// TwinCAT 3 PLC project PID_Projekt
// ProgramVersion: 3.1.4023.0
// libraries:
//   Tc2_ControllerToolbox, * (Beckhoff Automation GmbH)
//   Tc2_MC2, * (Beckhoff Automation GmbH)
//   Tc2_Standard, * (Beckhoff Automation GmbH)
//   Tc2_System, * (Beckhoff Automation GmbH)
//   Tc3_Module, * (Beckhoff Automation GmbH)
// project tree:
//   DUTs/ state.TcDUT
//   / GlobalTextList.TcGTLO, PID_Task.TcTTO, PlcTask.TcTTO
//   GVLs/ GVL.TcGVL
//   POUs/ MAIN.TcPOU
//   POUs/PID/ PID_Call.TcPOU, PRG_FB_CTRL_D.TcPOU, PRG_FB_CTRL_I.TcPOU, PRG_FB_CTRL_P.TcPOU
// real-time tasks:
//   TASK PlcTask: cycle T#1ms, priority 2, ADS port 350
//   TASK PID_Task: cycle T#10ms, priority 3, ADS port 351
// motion (NC):
//   TASK NC-Task 1 SAF: cycle T#1ms, priority 1, ADS port 501
//   TASK NC-Task 1 SVB: cycle T#10ms, priority 8, ADS port 511
//   AXIS Achse 1 (id 1) // MyAxis
//     Dynamic: Acceleration=3000, Deceleration=500
//     OtherSettings: AllowMotionCmdToSlave=true
//     encoder EncType=1
//     drive DrvType=5
//       Analog: TorqueSetpointScale=10, ScaleFactorActTorque=0.1
//       TimeComp: TaskDelayCycles=1
//     controller CtrType=1
//       CtrPara: PriorControlFactor=1
//         Observer: BandWidth=20
// variable links:
//   PID_Projekt/PID_Projekt Instance <-> NC-Task 1 SAF/Axes/Achse 1
//     PlcTask Inputs/MAIN.axis.NcToPlc <-> Outputs/ToPlc
//     PlcTask Outputs/MAIN.axis.PlcToNc <-> Inputs/FromPlc

CONFIGURATION PID_Projekt
    RESOURCE PLC ON TwinCAT3
        TASK PID_Task(INTERVAL := T#10ms, PRIORITY := 3);
        TASK PlcTask(INTERVAL := T#1ms, PRIORITY := 2);
        PROGRAM PID_Call WITH PID_Task : PID_Call;
        PROGRAM MAIN WITH PlcTask : MAIN;
    END_RESOURCE
END_CONFIGURATION

// ---- DUTs/state.TcDUT
TYPE state :
(
	INIT,
	POWER_ON,
	MOVE_ON,
	//MOVE_ON_NEWTARGETPOSITION,
	ERROR,
	P_RESET
)UDINT;
END_TYPE

// ---- GVLs/GVL.TcGVL
{attribute 'qualified_only'}
VAR_GLOBAL
	Signal: LREAL;
	Position: LREAL;
	Velocity: LREAL;
	Sollkraft: LREAL := 1;
	ErrorTerm: LREAL;
	PID_Output: LREAL;
	P_Regler: LREAL;
	I_Regler: LREAL;
	D_Regler: LREAL;
END_VAR

// ---- POUs/PID/PID_Call.TcPOU
PROGRAM PID_Call
VAR
	Simulation: BOOL := 0;
	Stoerungen: LREAL;
	SteadyState: BOOL := 0;
	D_Regler_Switch: BOOL := 1;
	I_Regler_Switch: BOOL := 1;
	Kp: LREAL;
	Satuaration_Check_LimMax: LREAL := 0.5;
	Satuaration_Check_LimMin: LREAL := -0.5;
	Not_Equal_Block: BOOL;
	Equal_Block: BOOL;
	PID_Output_after_S_check: LREAL;
	Drand: DRAND;
	PID_OUT_LimMin: LREAL := -0.9;
	PID_OUT_LimMax: LREAL := 0.9;
END_VAR

//*********Sensor
Drand(Seed:=0);
Stoerungen := (Drand.Num-0.5)*0.02;
GVL.Position := GVL.Position * (1+Stoerungen);
//GVL.Signal := GVL.Position;

//*********Error Term from Feedback Path
Drand(Seed:=0);	
Stoerungen := (Drand.Num-0.5)*0.02;
GVL.Signal := GVL.Position * (1+Stoerungen);
GVL.ErrorTerm := GVL.Sollkraft - GVL.Signal;

IF GVL.Position<(GVL.Sollkraft+0.015) AND GVL.Position>(GVL.Sollkraft-0.015) THEN
	SteadyState :=1;
ELSE SteadyState :=0;
END_IF

IF Simulation = 1 THEN
	GVL.ErrorTerm := GVL.Sollkraft - GVL.Signal * (1+(Drand.Num-0.5)*1);
END_IF

IF SteadyState = 0 THEN
	GVL.ErrorTerm := GVL.Sollkraft - GVL.Position;
	D_Regler_Switch := 0;
ELSE
//	GVL.ErrorTerm := GVL.Sollkraft - GVL.Signal;
	D_Regler_Switch := 1;
END_IF

//************I-Regler
PRG_FB_CTRL_P();

//************I-Regler
IF I_Regler_Switch=1 THEN			
	PRG_FB_CTRL_I();
END_IF

//************D-Regler (band-limited differentiator)
IF I_Regler_Switch=1 THEN
	PRG_FB_CTRL_D();
END_IF

//************Compute output and apply limits
GVL.PID_Output := GVL.P_Regler + GVL.I_Regler + GVL.D_Regler;

//************Saturation check
IF GVL.PID_Output > Satuaration_Check_LimMax THEN
	PID_Output_after_S_check := Satuaration_Check_LimMax;
ELSIF GVL.PID_Output < Satuaration_Check_LimMin THEN
	PID_Output_after_S_check := Satuaration_Check_LimMin;
END_IF

//************I-Regler Clamping
IF GVL.PID_Output = PID_Output_after_S_check THEN
	Not_Equal_Block:=0;
ELSE Not_Equal_Block:=1;
END_IF

IF ((GVL.PID_Output>0) AND (GVL.ErrorTerm>0)) OR ((GVL.PID_Output<0) AND (GVL.ErrorTerm<0)) OR ((GVL.PID_Output=0) AND (GVL.ErrorTerm=0))THEN
	Equal_Block := 1;
ELSE Equal_Block := 0;
END_IF

IF Not_Equal_Block AND Equal_Block THEN
	I_Regler_Switch := 0;
ELSE I_Regler_Switch := 1;
END_IF

END_PROGRAM

// ---- POUs/PID/PRG_FB_CTRL_P.TcPOU
PROGRAM PRG_FB_CTRL_P
VAR
	fIn								: LREAL					:= 15.0;
	fOut							: LREAL;

	eMode							: E_CTRL_MODE;
	stCTRL_P_PARAMS					: ST_CTRL_P_PARAMS;

	eErrorId						: E_CTRL_ERRORCODES;
	bError							: BOOL;

	(* controller *)
	fbCTRL_P						: FB_CTRL_P;

	bInit							: BOOL	:= TRUE;
	fbTON							: TON;
END_VAR

IF bInit THEN
	(* init parameter struct *)
	stCTRL_P_PARAMS.tCtrlCycleTime	:= T#10MS;
	stCTRL_P_PARAMS.tTaskCycleTime	:= T#10ms;
	stCTRL_P_PARAMS.fKp				:= 3;								(* gain Kp	*)

	(* set the mode to ACTIVE --> normal operation *)
	eMode	:= eCTRL_MODE_ACTIVE;

	(* reset the init flag *)
	bInit	:= FALSE;
END_IF


(* call controller *)
fbCTRL_P(fIn		:= GVL.ErrorTerm,
		 eMode		:= eMode,
		 stParams	:= stCTRL_P_PARAMS,
		 fOut		=> GVL.P_Regler,
		 eErrorId	=> eErrorId,
		 bError		=> bError);

END_PROGRAM

// ---- POUs/PID/PRG_FB_CTRL_I.TcPOU
PROGRAM PRG_FB_CTRL_I
VAR
	fIn								: LREAL					:= 15.0;
	fOut							: LREAL;

	eMode							: E_CTRL_MODE;
	stCTRL_I_PARAMS					: ST_CTRL_I_PARAMS;

	eErrorId						: E_CTRL_ERRORCODES;
	bError							: BOOL;

	(* controller *)
	fbCTRL_I						: FB_CTRL_I;

	bInit							: BOOL	:= TRUE;
	fbTON							: TON;
END_VAR

IF bInit THEN
	(* init parameter struct *)
	stCTRL_I_PARAMS.tCtrlCycleTime		:= T#10ms;
	stCTRL_I_PARAMS.tTaskCycleTime		:= T#10ms;
	stCTRL_I_PARAMS.tTi					:= T#2s;
	stCTRL_I_PARAMS.fOutMaxLimit		:=  10;
	stCTRL_I_PARAMS.fOutMinLimit		:= -10;

	(* set the mode to ACTIVE --> normal operation *)
	eMode := eCTRL_MODE_ACTIVE;

	(* reset the init flag *)
	bInit := FALSE;
END_IF


(* call controller *)
fbCTRL_I(	fIn					:= GVL.ErrorTerm,
			eMode				:= eMode,
			stParams			:= stCTRL_I_PARAMS,
			fOut				=> GVL.I_Regler,
			eErrorId			=> eErrorId,
			bError				=> bError);

END_PROGRAM

// ---- POUs/PID/PRG_FB_CTRL_D.TcPOU
PROGRAM PRG_FB_CTRL_D
VAR
	fIn						: LREAL					:= 10.0;
	fOut					: LREAL;

	fManSyncValue			: LREAL;
	bSync					: BOOL;

	eMode					: E_CTRL_MODE;
	stCTRL_D_PARAMS			: ST_CTRL_D_PARAMS;

	eErrorId				: E_CTRL_ERRORCODES;
	bError					: BOOL;
	(* controller *)
	fbCTRL_D				: FB_CTRL_D;
	
	bInit					: BOOL	:= TRUE;
	fbTON					: TON;
END_VAR

IF bInit THEN
	(* init parameter struct *)
	stCTRL_D_PARAMS.tCtrlCycleTime		:= T#10ms;
	stCTRL_D_PARAMS.tTaskCycleTime		:= T#10MS;
	stCTRL_D_PARAMS.tTv					:= T#0.01S;
	stCTRL_D_PARAMS.tTd					:= T#1S;
	stCTRL_D_PARAMS.fOutMaxLimit		:=  80.0;
	stCTRL_D_PARAMS.fOutMinLimit		:= -80.0;

	(* set the mode to ACTIVE --> normal operation *)
	eMode := eCTRL_MODE_ACTIVE;

	(* reset the init flag *)
	bInit := FALSE;
END_IF


(* call controller *)
fbCTRL_D	(	fIn					:= GVL.ErrorTerm,
				fManSyncValue		:= fManSyncValue,
				bSync				:= bSync,
				eMode				:= eMode,
				stParams			:= stCTRL_D_PARAMS,
				fOut				=> GVL.D_Regler,
				eErrorId			=> eErrorId,
				bError				=> bError
			);

END_PROGRAM

// ---- POUs/MAIN.TcPOU
PROGRAM MAIN
VAR
	MC_ReadActualVelocity: MC_ReadActualVelocity;
	state: state;
	
	reset_output:ST_McOutputs;
	axis_Reset: MC_Reset;
	ReadP_Valid:BOOL;
	ReadV_Valid:BOOL;
	power1: MC_Power;
	
	power1_output:ST_McOutputs;
	
    axis: AXIS_REF;
	StartInit: BOOL := 1;
	MC_MoveVelocity_0: MC_MoveVelocity;
	
	MoveVelocity_output:ST_McOutputs;
	MC_MoveVelocity_1: MC_MoveVelocity;
	MC_ReadActualPosition: MC_ReadActualPosition;
END_VAR

// Programmablauf mittels Zustandsautomat
CASE state OF
	
	INIT:
		MC_MoveVelocity_0.Execute := FALSE;
		Power1.Enable:=FALSE;
		axis_Reset.Execute := FALSE;
		state := POWER_ON;
		
	POWER_ON:
		Power1.Enable := TRUE;
		IF power1.Status THEN
				state := MOVE_ON;
		ELSIF power1.Error THEN
				state := ERROR;
		END_IF

	MOVE_ON:
		
		IF GVL.PID_Output>=0 THEN
			MC_MoveVelocity_0.Direction := MC_Positive_Direction;
			GVL.Velocity := GVL.PID_Output;
		ELSIF GVL.PID_Output<0 THEN
			MC_MoveVelocity_0.Direction := MC_Negative_Direction;
			GVL.Velocity := (-1) * GVL.PID_Output;
		ELSE MC_MoveVelocity_0.Direction := MC_Undefined_Direction;
		END_IF

		
		MC_MoveVelocity_0.Execute := TRUE;
		IF MoveVelocity_output.Done THEN
			MC_MoveVelocity_0.Execute := FALSE;
			state := MOVE_ON;
		ELSIF MC_MoveVelocity_0.CommandAborted OR MC_MoveVelocity_0.Error THEN
			state := ERROR;
		END_IF
		
	ERROR:
		IF axis.Status.Error THEN
			state := P_RESET;	(* axis error requires reset *)
		ELSE
			state := INIT;		(* function block errors don't need a reset *)
		END_IF
		
	P_RESET:
		axis_Reset.Execute := TRUE;
		MC_MoveVelocity_0.Execute := FALSE;
		IF axis_Reset.Done  THEN
			state := INIT;
		ELSIF axis_Reset.Error  THEN
			state := INIT; 
		END_IF
END_CASE

axis();
Power();
ActMove();
ReadP_V();
Reset();

ACTION ActMove:
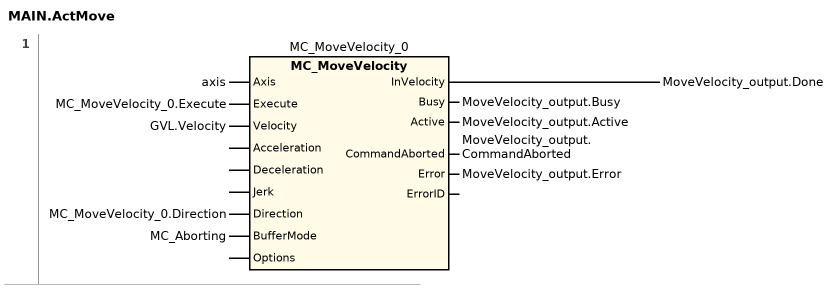
// NETWORK 1
MC_MoveVelocity_0(
    Axis := axis,
    Execute := MC_MoveVelocity_0.Execute,
    Velocity := GVL.Velocity,
    Direction := MC_MoveVelocity_0.Direction,
    BufferMode := MC_Aborting,
    Busy => MoveVelocity_output.Busy,
    Active => MoveVelocity_output.Active,
    CommandAborted => MoveVelocity_output.CommandAborted,
    Error => MoveVelocity_output.Error); // MC_MoveVelocity
MoveVelocity_output.Done := MC_MoveVelocity_0.InVelocity;
END_ACTION

ACTION Power:
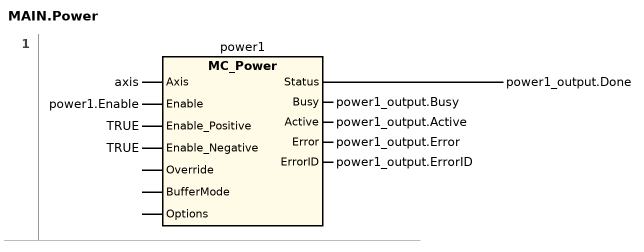
// NETWORK 1
power1(
    Axis := axis,
    Enable := power1.Enable,
    Enable_Positive := TRUE,
    Enable_Negative := TRUE,
    Busy => power1_output.Busy,
    Active => power1_output.Active,
    Error => power1_output.Error,
    ErrorID => power1_output.ErrorID); // MC_Power
power1_output.Done := power1.Status;
END_ACTION

ACTION ReadP_V:
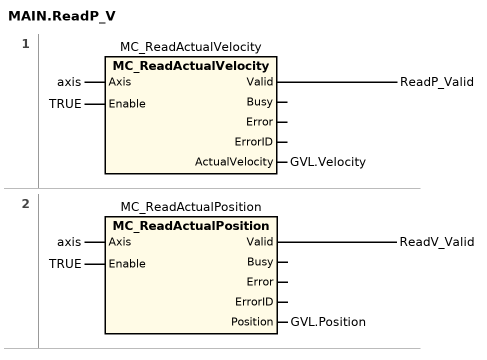
// NETWORK 1
MC_ReadActualVelocity(Axis := axis, Enable := TRUE, ActualVelocity => GVL.Velocity);
ReadP_Valid := MC_ReadActualVelocity.Valid;

// NETWORK 2
MC_ReadActualPosition(Axis := axis, Enable := TRUE, Position => GVL.Position);
ReadV_Valid := MC_ReadActualPosition.Valid;
END_ACTION

ACTION Reset:
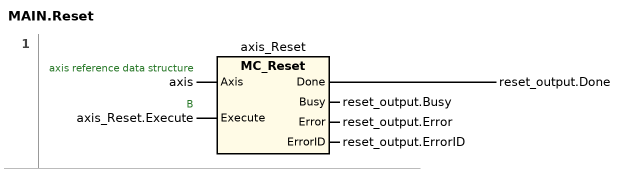
// NETWORK 1
//   axis: axis reference data structure
//   axis_Reset.Execute: B
axis_Reset(
    Axis := axis,
    Execute := axis_Reset.Execute,
    Busy => reset_output.Busy,
    Error => reset_output.Error,
    ErrorID => reset_output.ErrorID); // MC_Reset
reset_output.Done := axis_Reset.Done;
END_ACTION

END_PROGRAM

// ---- GlobalTextList.TcGTLO
TEXTLIST GlobalTextList
  95 = 'PowerEnable'
END_TEXTLIST
